FUNCTION_BLOCK ABSTRACT Xts IMPLEMENTS I_Cyclic, I_Initialisable, I_XTS, I_Object
VAR
	MyName : STRING;
	_MyXts : INT;
	_XtsEnabled : BOOL;
	_XPU : I_TcIoXtsProcessingUnit;
	_MoverArray : ARRAY[0..MaxMovers] OF I_XtsMover;
	_XtsIoEnvVar : I_XtsIoEnvVar;
	ICollisionGroup : I_CollisionGroup;
	_MyXtsHardware : I_XtsHardware;
	XtsHwState : XtsSystemInitialisation;
	EnableSequence : XtsEnableSequence;
	DisableSequence : XtsDisableSequence;	
	_Initialised : BOOL;
	EnabledTrigger : R_TRIG;
	DisabledTrigger : R_TRIG;
	_registeredNumberOfMovers: INT;
	DetectedMoverCount : UDINT;
	HardwareError : BOOL;
	CAGroupError : BOOL;
	_ErrorID : UDINT;
END_VAR
VAR CONSTANT
	MaxMovers : INT := 255;
END_VAR

{analysis -2}

METHOD AreAllMoversStationary : BOOL
VAR
	i : INT;
END_VAR
AreAllMoversStationary := TRUE;
FOR i := 0 TO _registeredNumberOfMovers - 1 DO
	IF NOT _MoverArray[i].IsStationary THEN
		AreAllMoversStationary := FALSE;
		EXIT;
	END_IF
END_FOR
END_METHOD

METHOD PUBLIC Cycle : HRESULT
VAR
	EnableResult : HRESULT;
	DisableResult : HRESULT;
	GrpStopResult : HRESULT;
	CollisionResult : HRESULT;
END_VAR
IF NOT _Initialised THEN	
	Cycle  := -1;
	RETURN;
END_IF

EnableResult := EnableSequence.Cycle();
DisableResult := DisableSequence.Cycle();
EnabledTrigger(CLK := EnableSequence.Done);
DisabledTrigger(CLK := DisableSequence.Done);
IF EnabledTrigger.Q THEN
	_XtsEnabled := TRUE;
END_IF
IF DisabledTrigger.Q THEN
	_XtsEnabled := false;
END_IF

HardwareError := _MyXtsHardware.AnyPartsInError;
CAGroupError := ICollisionGroup.HasError;

IF CAGroupError THEN
	_ErrorID := ICollisionGroup.ErrorCode;
END_IF
IF HardwareError THEN
	_ErrorID := _MyXtsHardware.GetPartErrorCode();
END_IF
IF NOT CAGroupError AND NOT HardwareError THEN
	_ErrorID := 0;
END_IF
END_METHOD

METHOD DisableXTS : BOOL
VAR_INPUT
END_VAR
IF _XtsEnabled THEN
	Base_Library.Tracing.Trace.Verbose(MyName, 'Disable Accepted');
	DisableXTS := SUCCEEDED(DisableSequence.Disable());
END_IF
END_METHOD

METHOD EnableXTS : BOOL
VAR_INPUT
END_VAR
IF NOT _XtsEnabled THEN
	Base_Library.Tracing.Trace.Verbose(MyName, 'Enable Accepted');
	EnableXts := SUCCEEDED(EnableSequence.Enable());
END_IF
END_METHOD

PROPERTY ErrorId : UDINT
GET
_ErrorID := _ErrorID;
END_GET
END_PROPERTY

PROPERTY ExpectedNumberOfParts : int
GET
ExpectedNumberOfParts := _MyXtsHardware.ExpectedNumberOfParts;
END_GET
SET
_MyXtsHardware.ExpectedNumberOfParts := ExpectedNumberOfParts;
END_SET
END_PROPERTY

PROPERTY ExpectedNumberOfTracks : int
GET
ExpectedNumberOfTracks := _MyXtsHardware.ExpectedNumberOfTracks;
END_GET
SET
_MyXtsHardware.ExpectedNumberOfTracks := ExpectedNumberOfTracks;
END_SET
END_PROPERTY

//FB_Init is always available implicitly and it is used primarily for initialization.
//The return value is not evaluated. For a specific influence, you can also declare the
//methods explicitly and provide additional code there with the standard initialization
//code. You can evaluate the return value.
METHOD FB_Init: BOOL
VAR_INPUT
    bInitRetains: BOOL; // TRUE: the retain variables are initialized (reset warm / reset cold)
    bInCopyCode: BOOL;  // TRUE: the instance will be copied to the copy code afterward (online change)   
	MyXtsIoEnvVar : I_XtsIoEnvVar;
	MyXtsHardware : I_XtsHardware;
	MyCAGroup : I_CollisionGroup;
END_VAR
_XtsIoEnvVar := MyXtsIoEnvVar;
_MyXtsHardware := MyXtsHardware;
ICollisionGroup := MyCAGroup;
EnableSequence.MyCollisionGroup := ICollisionGroup;
DisableSequence.MyCollisionGroup := ICollisionGroup;
END_METHOD

PROPERTY HasError : BOOL
GET
HasError := ICollisionGroup.HasError OR _MyXtsHardware.AnyPartsInError;
END_GET
END_PROPERTY

METHOD Initialise : HRESULT
VAR
	i : INT;
END_VAR
Initialise := -1;
CASE XtsHwState OF
	XtsSystemInitialisation.WaitingForXtsIoEnvVar:
		IF _XtsIoEnvVar.Initialised THEN
			_XPU := _XtsIoEnvVar.GetXPUInterface(_MyXts);
			_MyXtsHardware.MyXpu := _XPU;
			XtsHwState := XtsSystemInitialisation.PassGroupReference;
		END_IF
		
	XtsSystemInitialisation.PassGroupReference:
		ICollisionGroup.CAGroupXtsIoEnvInterface := _XtsIoEnvVar.GetCaGroupInterface(_MyXts);
		XtsHwState := XtsSystemInitialisation.WaitingForHardwareToInitialise;
	
	XtsSystemInitialisation.WaitingForHardwareToInitialise:
		IF _MyXtsHardware.Initialised THEN
			MyName := _MyXtsHardware.MyName;
			XtsHwState := XtsSystemInitialisation.SetATrackForDetection;
		END_IF
	
	XtsSystemInitialisation.SetATrackForDetection:
		IF SUCCEEDED(_MyXtsHardware.SetATrackForDetection(1)) THEN
			XtsHwState := XtsSystemInitialisation.TriggeringRedetection;
		END_IF
		
	XtsSystemInitialisation.TriggeringRedetection:
		IF SUCCEEDED(_MyXtsHardware.TriggerMoverRedetection()) THEN
			XtsHwState := XtsSystemInitialisation.WaitingForAllMoversValid;
		END_IF
		
	XtsSystemInitialisation.WaitingForAllMoversValid:
		IF _MyXtsHardware.AllMoverPositionsValid THEN
			XtsHwState := XtsSystemInitialisation.CheckingAllMoverFound;
		END_IF
	
	XtsSystemInitialisation.CheckingAllMoverFound:
		IF _MyXtsHardware.AreExpectedMoversFound() THEN
			DetectedMoverCount := _MyXtsHardware.NumberOfMoversDetected;
			XtsHwState := XtsSystemInitialisation.CheckIfXtsInSimMode;
		END_IF
		
	XtsSystemInitialisation.CheckIfXtsInSimMode:
		IF _MyXtsHardware.XtsInSim THEN
			XtsHwState := XtsSystemInitialisation.TriggeringMoverIdDetection;
		ELSE
			XtsHwState := XtsSystemInitialisation.CheckingXts24And48Volts;
		END_IF
		
	XtsSystemInitialisation.CheckingXts24And48Volts:
		IF SUCCEEDED(_MyXtsHardware.IsHardware24VdcOK()) AND SUCCEEDED(_MyXtsHardware.IsHardware48VdcOK()) THEN
			XtsHwState := XtsSystemInitialisation.TriggeringMoverIdDetection;
		END_IF
	
	XtsSystemInitialisation.TriggeringMoverIdDetection:
		IF _MyXtsHardware.IsIDDetectionStandard() OR_ELSE SUCCEEDED(_MyXtsHardware.TriggerMoverIDDetection()) THEN
			XtsHwState := XtsSystemInitialisation.XtsInitialised;
		END_IF
	
	XtsSystemInitialisation.XtsInitialised:
		Initialise := 0;
		_Initialised := TRUE;	
END_CASE
END_METHOD

PROPERTY Initialised : BOOL
GET
Initialised := _Initialised;
END_GET
END_PROPERTY

PROPERTY IsIdle : BOOL
GET
IsIdle := DisableSequence.Done;
END_GET
END_PROPERTY

PROPERTY IsReady : BOOL
GET
IsReady := _XtsEnabled;
END_GET
END_PROPERTY

METHOD PUBLIC Abstract MoverHomeSequence : BOOL
VAR_INPUT
END_VAR
END_METHOD

PROPERTY MyXts : INT
GET
MyXts := _MyXtsHardware.MyXts;
END_GET
SET
_MyXtsHardware.MyXts := _MyXts := MyXts;
END_SET
END_PROPERTY

METHOD RegisterMovers : HRESULT
VAR_INPUT
	MyMover : I_XtsMover;
END_VAR
VAR
	i : UINT;
	MoverRegistered: BOOL;
END_VAR
IF MyMover = 0 THEN
	Base_Library.Tracing.Trace.Warning(MyName, 'Register Mover Fail - null ptr');
	RegisterMovers := -1;
	RETURN;
END_IF
IF NOT _Initialised THEN
	Base_Library.Tracing.Trace.Warning(MyName, 'Register Mover Fail - not ready');
	RegisterMovers := -2;
	RETURN;
END_IF
IF _registeredNumberOfMovers >= MaxMovers THEN
	Base_Library.Tracing.Trace.Warning(MyName, 'Register Mover Fail - max movers reached');
	RegisterMovers := -3;
	RETURN;
END_IF
FOR i := 0 TO (_registeredNumberOfMovers - 1) DO
	IF _MoverArray[i] = MyMover THEN
		MoverRegistered := TRUE;
		EXIT;
	END_IF
END_FOR
IF MoverRegistered THEN
	Base_Library.Tracing.Trace.Warning(MyName, 'Register Mover Fail - registered');
	RegisterMovers := -4;
	RETURN;
END_IF

Base_Library.Tracing.Trace.Verbose(MyName, 'Register Mover Accepted');
_MoverArray[_registeredNumberOfMovers] := MyMover;
_registeredNumberOfMovers := _registeredNumberOfMovers + 1;
EnableSequence.RegisterMovers(MyMover);
DisableSequence.RegisterMovers(MyMover);
FOR i := 1 TO _MyXtsHardware.DetectedNumberOfTracks DO
	MyMover.RegisterTracks(Track := _MyXtsHardware.GetTrackInterfaceByNumber(i));
END_FOR
FOR i := 1 TO TO_UINT(_XPU.GetDetectedMoverCount()) DO
	IF MyMover.AxisRef.NcToPlc.AxisId = _XPU.MoverTcIo(i).P_AxisId THEN
		MyMover.MoverXtsIoEnvInterface := _XPU.MoverTcIo(i);
	END_IF
END_FOR
END_METHOD

METHOD RegisterWithParent
VAR_INPUT
	Parent	: I_HostObjects;
END_VAR
Parent.RegisterCyclic(THIS^);
Parent.RegisterInitialisable(THIS^);
END_METHOD

METHOD Reset : BOOL
VAR_INPUT
END_VAR
Reset := SUCCEEDED(ICollisionGroup.Reset());
_MyXtsHardware.ResetAllParts();
Base_Library.Tracing.Trace.Verbose(MyName, 'Reset Accepted');
END_METHOD

METHOD StopXts : BOOL
VAR_INPUT
END_VAR
StopXTS := ICollisionGroup.GroupStop();
Base_Library.Tracing.Trace.Verbose(MyName, 'Stop Accepted');
END_METHOD

END_FUNCTION_BLOCK

(* stored: Version 1.1.0.1
   POU Xts: Id {4538c683-94fc-49a1-b5ad-30ffec5e4eff}, SpecialFunc None
   Folder Operations: Id {0e8598c4-3d58-4c14-a12f-6fd3f3ea02bf}
   Folder Settings: Id {cec05bdb-9232-4b5d-b91e-848bd7bc55d9}
   Folder Status: Id {c34f5481-c408-4671-a299-9c4a6e31956c}
   Method AreAllMoversStationary: Id {f009ccd3-c388-424a-b98d-ae435064fa0b}
   Method Cycle: Id {da42838e-fb00-40a5-96f4-b787aa883566}
   Method DisableXTS: Id {e2a85e5a-c7bf-481d-be4f-81acebc29fb7}
   Method EnableXTS: Id {e800781e-1435-4747-9cb4-9b9fab34ca22}
   Property ErrorId: Id {d9cfe84c-7a4b-4b34-a9ba-97d2ea994ecf}
   Get Get: Id {052b70ff-e616-4a6d-a158-86a46066c230}
   Property ExpectedNumberOfParts: Id {33632734-2180-4c77-982d-f6997ead5bb5}
   Get Get: Id {ec285ff9-810a-46b0-8941-68dcdc1ab79d}
   Set Set: Id {4cb5fde4-6845-43ef-b95e-df4929829b0c}
   Property ExpectedNumberOfTracks: Id {6b69c4c6-afe3-46d9-bc08-86224f82f24a}
   Get Get: Id {cab0d03f-ccb1-4d2e-adb6-3d697ceee44c}
   Set Set: Id {b24fc04c-e333-4935-bdff-3eff5a7d9932}
   Method FB_Init: Id {d6ce6c85-5c43-4276-b07f-92a2e669b228}
   Property HasError: Id {fc5d4c9f-c257-47d7-8282-ec3a9f63c6e5}
   Get Get: Id {e073db15-e4f5-4f0c-b72a-f5365dbb2c5c}
   Method Initialise: Id {3c52ae7d-89c5-4979-a1bd-5023a279947c}
   Property Initialised: Id {a78fe92f-7cf8-4747-affa-2e0853d05d4c}
   Get Get: Id {8057f725-8638-4356-89d5-da5eb20cf86c}
   Property IsIdle: Id {3c144ba6-395b-4ea8-98ac-f2364ab509f3}
   Get Get: Id {e2c9271f-6b55-4d9e-90f5-2964294aa055}
   Property IsReady: Id {2e2a3eb7-41f9-4889-9a54-93f51d339119}
   Get Get: Id {c1a60130-732b-467c-8f85-c88373ac5c2c}
   Method MoverHomeSequence: Id {5c2deb91-ebd0-4a93-99ec-6a6bbbd5e076}
   Property MyXts: Id {b982f888-fcea-49f3-8b85-76339b257fce}
   Get Get: Id {7260ae55-6d72-4286-9779-c205f4bf658b}
   Set Set: Id {f9bbe24a-eac8-4b47-a949-a650212b0818}
   Method RegisterMovers: Id {a3bbc877-121f-4130-8916-a04d2ba4dd9d}
   Method RegisterWithParent: Id {5a27c335-0022-4ddf-98ff-1436953bbdbd}
   Method Reset: Id {f4cda3e0-308c-460d-87ee-c1616441d1b6}
   Method StopXts: Id {4b648283-f5f4-4d47-a58f-be53e519365d} *)
